// TIA Portal project "TS_Stoliar_DP" (V20)

(* hardware
DEVICE "S7-1200 G2 station_1"  S7-1200 G2 Station
   slot 0: "Rack_0"  S71200G2 Rack  Rack  V1.0
   slot 1: "G2_PLC_1"  CPU 1214C DC/DC/DC  6ES7 214-1AH50-0XB0  V1.0
   slot 9: "AI2/AQ2 signal board_1"  AI2/AQ2 signal board  6ES7 233-4HD50-0XB0  V1.0
*)

// ===== PLC "G2_PLC_1"  CPU 1214C DC/DC/DC =====

VAR_GLOBAL   // PLC tag table "Default tag table"
   "VENT" AT %QW80 : Int;
   "SPIR" AT %QW82 : Int;
   "Tag_3" AT %IW80 : Int;
   "Tag_4" AT %IW82 : Int;
END_VAR

DATA_BLOCK "DATA"   // DB1
{ S7_Optimized_Access := 'TRUE' }
VERSION : 0.1
   VAR
      y : Real;
      u : Real;
      vent : Real;
   END_VAR
BEGIN
END_DATA_BLOCK

FUNCTION_BLOCK "FB_PI_TS05"   // FB1, SCL
{ S7_Optimized_Access := 'TRUE' }
VERSION : 0.1
   VAR_INPUT
      Y : Real;
      Setpoint_pb : Real;
      Enable : Bool;
      Reset : Bool;
      TimeSec : Real;
   END_VAR
   VAR_OUTPUT
      U : Real;
      DU : Real;
      "E" : Real;
      Ypb_out : Real;
      Integrator_out : Real;
   END_VAR
   VAR
      Integrator : Real;
      Ypb : Real;
      Started : Bool;
   END_VAR
   VAR CONSTANT
      Kp : Real := 3.58;
      Ki : Real := 1.84;
      Ts : Real := 0.1;
      U_pb : Real := 4.0;
      DU_min : Real := -4.0;
      DU_max : Real := 6.0;
   END_VAR
BEGIN
   IF #Reset THEN
       #Integrator := 0.0;
       #Ypb := 0.0;
       #Started := FALSE;
       #U := #U_pb;
       #DU := 0.0;
       #E := 0.0;

   ELSIF NOT #Enable THEN
       #U := #U_pb;
       #DU := 0.0;
       #E := 0.0;

   ELSE
       IF #TimeSec < 600.0 THEN
           #U := #U_pb;
           #Integrator := 0.0;
           #Ypb := #Y;
           #Started := True;
           #DU := 0.0;
           #E := 0.0;
       ELSE
           #E := #Setpoint_pb - (#Y - #Ypb);
           #Integrator := #Integrator + #E * #Ts;
           #DU := #Kp * #E + #Ki * #Integrator;

           IF #DU > #DU_max THEN
               #DU := #DU_max;
           ELSIF #DU < #DU_min THEN
               #DU := #DU_min;
           END_IF;

           #U := #DU + #U_pb;
       END_IF;
   END_IF;

   #Ypb_out := #Ypb;
   #Integrator_out := #Integrator;
END_FUNCTION_BLOCK

ORGANIZATION_BLOCK "Main"   // OB1, LAD, ProgramCycle
TITLE = "Main Program Sweep (Cycle)"
{ S7_Optimized_Access := 'TRUE' }
VERSION : 0.1
   VAR_INPUT
      Initial_Call : Bool;   // Initial call of this OB
      Remanence : Bool;   // =True, if remanent data are available
   END_VAR
   VAR_TEMP
      temp_real : Real;
   END_VAR
BEGIN

REGION Network 2
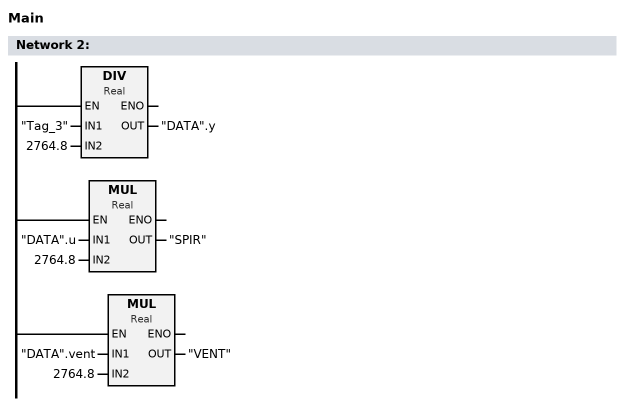
   RUNG wire#powerrail
      { S7_Templates := "SrcType := Real" } Div(in1 := "Tag_3", in2 := 2764.8, out => "DATA".y)
   END_RUNG
   RUNG wire#powerrail
      { S7_Templates := "SrcType := Real" } Mul(in1 := "DATA".u, in2 := 2764.8, out => "SPIR")
   END_RUNG
   RUNG wire#powerrail
      { S7_Templates := "SrcType := Real" } Mul(in1 := "DATA".vent, in2 := 2764.8, out => "VENT")
   END_RUNG
   // the same network as SCL:
   "DATA".y := "Tag_3" / 2764.8;
   "SPIR" := "DATA".u * 2764.8;
   "VENT" := "DATA".vent * 2764.8;
END_REGION
END_ORGANIZATION_BLOCK